PROGRAM MAIN
VAR
	stWash1 : ST_Wash := (nWaterLevel := 4, eWashStrategy := E_Strategy.SOFT );
	fbMotor : FB_BaseMotor;
	fbWaterController : FB_WaterController;
	fbWashingMachine : FB_WashingMachine( _iMotor := fbMotor, _iWaterController := fbWaterController );
	bStart: BOOL;
END_VAR

IF bStart THEN
	fbWashingMachine(stWash := stWash1);
END_IF

END_PROGRAM

(* stored: Version 1.1.0.1, ProductVersion 3.1.4024.16
   POU MAIN: Id {0dbc5495-60a6-448c-a4e7-d500a20e79f9}, SpecialFunc None *)
